// TIA Portal project "OhrevVody" (V15)

(* hardware
DEVICE "S71500/ET200MP station_1"  S7-1500 station
   slot 0: "Rail_0"  Rack  6ES7 590-1***0-0AA0
   slot 1: "PLCOhrev"  CPU 1515-2 PN  6ES7 515-2AM01-0AB0  V2.5
      slot 3: "CPU display_1"  6ES7591-1BA00-0AA0
   slot 2: "AQ 8xU/I HS_1"  AQ 8xU/I HS  6ES7 532-5HF00-0AB0  V2.1
   slot 3: "AI 8xU/I HF_1"  AI 8xU/I HF  6ES7 531-7NF00-0AB0  V1.1
   slot 4: "DI 16x24VDC BA_1"  DI 16x24VDC BA  6ES7 521-1BH10-0AA0  V1.0
*)

// ===== PLC "PLCOhrev"  CPU 1515-2 PN =====

VAR_GLOBAL   // PLC tag table "Default tag table"
   "P1" AT %QW0 : Int;
   "Horak" AT %QW2 : Int;
   "Teplota" AT %IW0 : Int;
   "ON" AT %I16.0 : Bool;
   "T2" AT %IW2 : Int;
END_VAR

DATA_BLOCK "Cerpadla_DB"   // DB1
{ S7_Optimized_Access := 'TRUE' }
VERSION : 0.1
// stored: InstanceOfName Cerpadla
"Cerpadla"
BEGIN
END_DATA_BLOCK

ORGANIZATION_BLOCK "Main"   // OB1, LAD, ProgramCycle
TITLE = "Main Program Sweep (Cycle)"
{ S7_Optimized_Access := 'TRUE' }
VERSION : 0.1
   VAR_INPUT
      Initial_Call : Bool;   // Initial call of this OB
      Remanence : Bool;   // =True, if remanent data are available
   END_VAR
   VAR_TEMP
      normTeplota : Real;
      teplota : Real;
   END_VAR
BEGIN

REGION Network 1
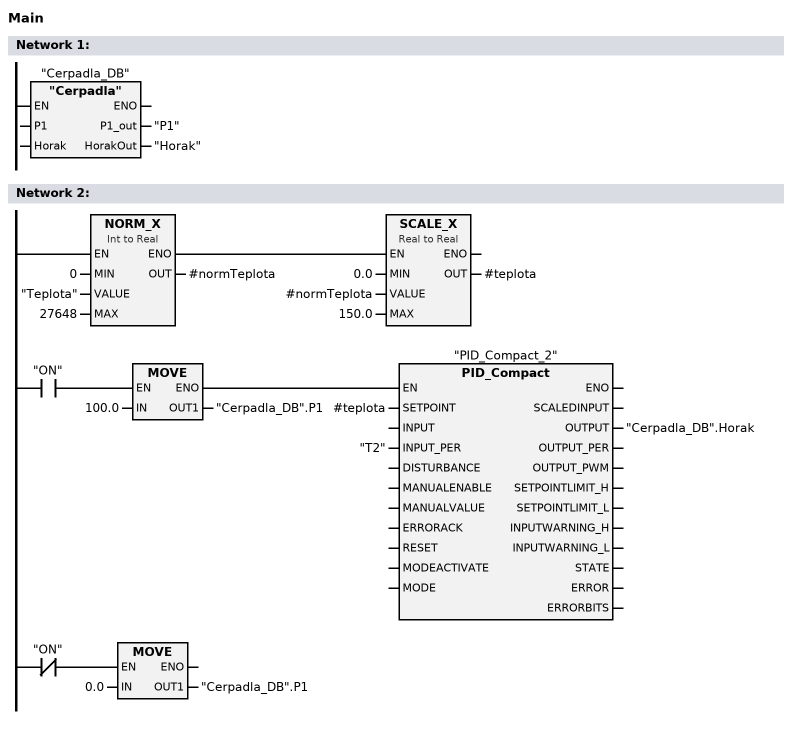
   RUNG wire#powerrail
      "Cerpadla_DB"(P1 :=, Horak :=, P1_out => "P1", HorakOut => "Horak")
   END_RUNG
   // the same network as SCL:
   "Cerpadla_DB"(P1_out => "P1", HorakOut => "Horak");   // "Cerpadla"
END_REGION

REGION Network 2
   #normTeplota := NORM_X(MIN := 0, VALUE := "Teplota", MAX := 27648);
   #teplota := SCALE_X(MIN := 0.0, VALUE := #normTeplota, MAX := 150.0);
   IF "ON" THEN
       "Cerpadla_DB".P1 := 100.0;
       "PID_Compact_2"(Setpoint := #teplota, Input_PER := "T2", Output => "Cerpadla_DB".Horak);   // PID_Compact
   END_IF;
   IF NOT "ON" THEN "Cerpadla_DB".P1 := 0.0; END_IF;
END_REGION
END_ORGANIZATION_BLOCK

// folder: Pristroje

FUNCTION_BLOCK "Cerpadla"   // FB1, LAD
{ S7_Optimized_Access := 'TRUE' }
VERSION : 0.1
   VAR_INPUT
      P1 : Real;
      Horak : Real;
   END_VAR
   VAR_OUTPUT
      P1_out : Int;
      HorakOut : Int;
   END_VAR
   VAR_TEMP
      normP1 : Real;
      normHorak : Real;
   END_VAR
BEGIN

REGION Network 1: P1
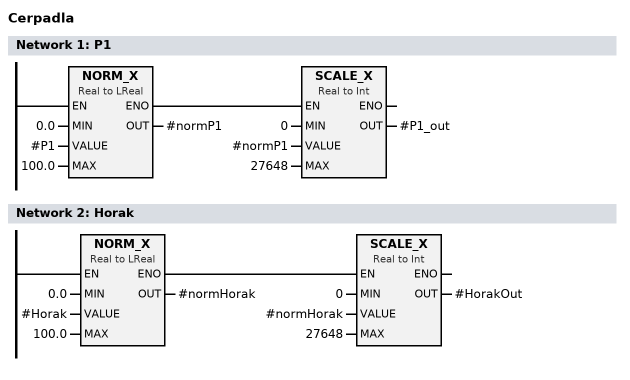
   RUNG wire#powerrail
      { S7_Templates := "[SrcType := Real, DestType := LReal]" } Normalize(min := 0.0, value := #P1, max := 100.0, out => #normP1)
      { S7_Templates := "[SrcType := Real, DestType := Int]" } Scale(min := 0, value := #normP1, max := 27648, out => #P1_out)
   END_RUNG
   // the same network as SCL:
   #normP1 := NORM_X(MIN := 0.0, VALUE := #P1, MAX := 100.0);
   #P1_out := SCALE_X(MIN := 0, VALUE := #normP1, MAX := 27648);
END_REGION

REGION Network 2: Horak
   RUNG wire#powerrail
      { S7_Templates := "[SrcType := Real, DestType := LReal]" } Normalize(min := 0.0, value := #Horak, max := 100.0, out => #normHorak)
      { S7_Templates := "[SrcType := Real, DestType := Int]" } Scale(min := 0, value := #normHorak, max := 27648, out => #HorakOut)
   END_RUNG
   // the same network as SCL:
   #normHorak := NORM_X(MIN := 0.0, VALUE := #Horak, MAX := 100.0);
   #HorakOut := SCALE_X(MIN := 0, VALUE := #normHorak, MAX := 27648);
END_REGION
END_FUNCTION_BLOCK